VAR_GLOBAL
	///input fb instance Cyl_AB position retract normally open
	In_bolHOR_2_Retracted_NO AT %I* : BOOL;
	///input fb instance Cyl_AB position extend normally closed
	In_bolHOR_2_Extended_NC AT %I*: BOOL;
	///output fb instance Cyl_AB valve retract
	Out_bolHOR_2_Retract AT %Q* : BOOL;
	///output fb instance Cyl_AB valve extend
	Out_bolHOR_2_Extend AT %Q* : BOOL;
END_VAR

(* stored: Version 1.1.0.1, ProductVersion 3.1.0.18
   GVL Io: Id {c2eadd2a-782d-4876-a2c7-8b2a9c7407cb} *)
